FUNCTION_BLOCK Pendulum4Tc
VAR_INPUT
	TimeSourceDateTime : I_PtTimesource;
END_VAR
VAR_OUTPUT
END_VAR
VAR
	_DateTime : PtDateTime;
	_Interval : PtInterval;
END_VAR


_DateTime := TimeSourceDateTime.getDateTime();

METHOD New : PtDateTime
VAR_INPUT
	Year : DINT;
	Month : DINT;
	Day : DINT;
	Hour : DINT;
	Minute : DINT;
	Second : DINT;
	Microsecond : DINT;
	TimeZone : DINT;
END_VAR
New.Set(
	Year:= Year, 
	Month:= Month, 
	Day:= Day, 
	Hour:= Hour, 
	Minute:= Minute, 
	Second:= Second, 
	Microsecond:= Microsecond, 
	TimeZone:= TimeZone);
END_METHOD

METHOD Now : PtDateTime
VAR_INPUT
END_VAR
Now := _DateTime;
END_METHOD

END_FUNCTION_BLOCK

(* stored: Version 1.1.0.1, ProductVersion 3.1.4024.12
   POU Pendulum4Tc: Id {e50634ac-d110-4401-be63-aef27cde4903}, SpecialFunc None
   Method New: Id {880ad30d-745b-4636-829f-cd855681e435}
   Method Now: Id {d16f0450-0a34-4f23-abde-57bf728c825e} *)
